// TIA Portal V19 export
DATA_BLOCK "acDataPointers"   // DB20
{ S7_Optimized_Access := 'TRUE' }
// stored: AutoNumber false, MemoryReserve 0
   VAR RETAIN
      ACT : "_AC_Interface";
      acInt : Array[0..31] of "_AC_Interface";   // Process Object pointers
   END_VAR
BEGIN
   acInt[0..4].ia.dbno := 27;
   acInt[0].ia.sta := 10;
   acInt[1].ia.sta := 1044;
   acInt[2].ia.sta := 2082;
   acInt[3].ia.sta := 3452;
   acInt[4].ia.sta := 5508;
   acInt[5].ia.sta := 4634;
   acInt[6].ia.sta := 6134;
   acInt[7].ia.sta := 7634;
   acInt[8].ia.sta := 9134;
   acInt[9].ia.sta := 10102;
   acInt[10].ia.sta := 11070;
   acInt[11].ia.sta := 12038;
   acInt[12].ia.sta := 13006;
   acInt[13].ia.sta := 314;
   acInt[14].ia.sta := 1178;
   acInt[15].ia.sta := 2042;
   acInt[17].ia.sta := 13974;
   acInt[18].ia.sta := 15062;
   acInt[19].ia.sta := 16030;
   acInt[20].ia.sta := 17530;
   acInt[21].ia.sta := 18498;
   acInt[22].ia.sta := 19466;
   acInt[23].ia.sta := 2906;
   acInt[24].ia.sta := 3770;
   acInt[25].ia.sta := 20460;
   acInt[0..1].ia.al := 1022;
   acInt[2].ia.al := 1346;
   acInt[3..4].ia.al := 2034;
   acInt[5..7].ia.al := 1226;
   acInt[8..12].ia.al := 962;
   acInt[13..15].ia.al := 858;
   acInt[17].ia.al := 1082;
   acInt[18].ia.al := 962;
   acInt[19].ia.al := 1226;
   acInt[20..22].ia.al := 962;
   acInt[23..24].ia.al := 858;
   acInt[25].ia.al := 962;
   acInt[0].IHW := 361;
   acInt[1].IHW := 362;
   acInt[2].IHW := 363;
   acInt[3].IHW := 364;
   acInt[4].IHW := 365;
   acInt[5].IHW := 352;
   acInt[6].IHW := 353;
   acInt[7].IHW := 354;
   acInt[8].IHW := 370;
   acInt[9].IHW := 371;
   acInt[10].IHW := 372;
   acInt[11].IHW := 373;
   acInt[12].IHW := 374;
   acInt[13].IHW := 375;
   acInt[14].IHW := 379;
   acInt[15].IHW := 380;
   acInt[16].IHW := 384;
   acInt[17].IHW := 388;
   acInt[18].IHW := 389;
   acInt[19].IHW := 390;
   acInt[20].IHW := 391;
   acInt[21].IHW := 392;
   acInt[22].IHW := 393;
   acInt[23].IHW := 394;
   acInt[24].IHW := 395;
   acInt[25].IHW := 355;
   acInt[0].IIp := 1;
   acInt[1].IIp := 2;
   acInt[2].IIp := 3;
   acInt[3].IIp := 4;
   acInt[4].IIp := 5;
   acInt[5].IIp := 1;
   acInt[6].IIp := 2;
   acInt[7].IIp := 3;
   acInt[8].IIp := 1;
   acInt[9].IIp := 2;
   acInt[10].IIp := 3;
   acInt[11].IIp := 4;
   acInt[12].IIp := 5;
   acInt[13].IIp := 6;
   acInt[14].IIp := 1;
   acInt[15].IIp := 2;
   acInt[16].IIp := 6;
   acInt[17].IIp := 1;
   acInt[18].IIp := 2;
   acInt[19].IIp := 3;
   acInt[20].IIp := 4;
   acInt[21].IIp := 5;
   acInt[22].IIp := 6;
   acInt[23].IIp := 7;
   acInt[24].IIp := 8;
   acInt[25].IIp := 5;
   acInt[0..4].op.dbno := 27;
   acInt[16].op.dbno := 0;
   acInt[0].op.sta := 4;
   acInt[1].op.sta := 1038;
   acInt[2].op.sta := 2076;
   acInt[3].op.sta := 3430;
   acInt[4].op.sta := 5486;
   acInt[5].op.sta := 4628;
   acInt[6].op.sta := 6128;
   acInt[7].op.sta := 7628;
   acInt[8].op.sta := 9128;
   acInt[9].op.sta := 10096;
   acInt[10].op.sta := 11064;
   acInt[11].op.sta := 12032;
   acInt[12].op.sta := 13000;
   acInt[13].op.sta := 308;
   acInt[14].op.sta := 1172;
   acInt[15].op.sta := 2036;
   acInt[17].op.sta := 13968;
   acInt[18].op.sta := 15056;
   acInt[19].op.sta := 16024;
   acInt[20].op.sta := 17524;
   acInt[21].op.sta := 18492;
   acInt[22].op.sta := 19460;
   acInt[23].op.sta := 2900;
   acInt[24].op.sta := 3764;
   acInt[25].op.sta := 20454;
   acInt[16].op.al := 0;
   acInt[0..4].cmds.dbno := 27;
   acInt[16].cmds.dbno := 0;
   acInt[0].cmds.sta := 6;
   acInt[1].cmds.sta := 1040;
   acInt[2].cmds.sta := 2078;
   acInt[3].cmds.sta := 3432;
   acInt[4].cmds.sta := 5588;
   acInt[5].cmds.sta := 4630;
   acInt[7].cmds.sta := 7630;
   acInt[8].cmds.sta := 9130;
   acInt[9].cmds.sta := 10098;
   acInt[10].cmds.sta := 11066;
   acInt[11].cmds.sta := 12034;
   acInt[12].cmds.sta := 13002;
   acInt[13].cmds.sta := 310;
   acInt[14].cmds.sta := 1174;
   acInt[15].cmds.sta := 2038;
   acInt[17].cmds.sta := 13970;
   acInt[18].cmds.sta := 15058;
   acInt[19].cmds.sta := 16026;
   acInt[20].cmds.sta := 17526;
   acInt[21].cmds.sta := 18494;
   acInt[22].cmds.sta := 19462;
   acInt[23].cmds.sta := 2902;
   acInt[24].cmds.sta := 3766;
   acInt[25].cmds.sta := 20456;
   acInt[16].cmds.al := 0;
   acInt[0..2].ev.dbno := 0;
   acInt[13..15].ev.dbno := 0;
   acInt[23].ev.dbno := 0;
   acInt[4].ev.sta := 10;
   acInt[5].ev.sta := 20;
   acInt[6].ev.sta := 30;
   acInt[7].ev.sta := 40;
   acInt[8].ev.sta := 50;
   acInt[9].ev.sta := 60;
   acInt[10].ev.sta := 70;
   acInt[11].ev.sta := 80;
   acInt[12].ev.sta := 90;
   acInt[16].ev.sta := 100;
   acInt[17].ev.sta := 110;
   acInt[18].ev.sta := 120;
   acInt[19].ev.sta := 130;
   acInt[20].ev.sta := 140;
   acInt[21].ev.sta := 150;
   acInt[22].ev.sta := 160;
   acInt[25].ev.sta := 170;
   acInt[0..2].ev.al := 0;
   acInt[13..15].ev.al := 0;
   acInt[23].ev.al := 0;
END_DATA_BLOCK
